Universal Robots PolyScope program: ad_lab_exe_4_2_64.urp

Program ad_lab_exe_4_2_64 (createdIn=3.2.19293 lastSavedIn=3.2.19293 directory=/programs installation=default robotSerialNumber=2015351391)
Calibrated DH parameters: a=[0.000352, -0.161198, -0.373486, 0.00005, 0.000049, 0]; d=[0.089268, 352.477598, -320.08558, -32.281492, 0.094939, 0.082518]; alpha=[1.570728, 0.001116, -0.003686, 1.571189, -1.570572, 0]; deltaTheta=[-0.000012, 1.181849, -1.491165, 0.309495, -0.000007, 0.000025]
Robot Program (runOnlyOnce=false motionType=MoveJ speed=1.047198 acceleration=1.396263 recalculateMotions=false)
  Folder 文件夹
    tcp1 := p[0,0,0.2,0,0,0]
    tcp2 := p[0.2,0,0.05,0,d2r(90),0]
    Script: set_tcp(tcp1)
    MoveL speed 250 mm/s, acceleration 1200 mm/s^2 (recalculateMotions=false) feature=Base
      Waypoint waypoint1: TCP in base x=137.871 y=664.13 z=276.516 mm, rx=-1.3493 ry=2.4374 rz=0.4077 rad; joints [96.893, -88.292, -94.384, -84.585, 94.191, -232.18] deg; flange x=46.759 y=487.114 z=417.839 mm, rx=1.522 ry=-2.6851 rz=-0.1148 rad
      Waypoint place_pos: TCP in base x=-60.021 y=25.367 z=248.738 mm, rx=0.8568 ry=-1.3626 rz=0.7366 rad; joints [108.205, -40.851, -138.273, -87.315, 93.558, -220.796] deg; flange x=46.759 y=195.075 z=296.65 mm, rx=1.522 ry=-2.6851 rz=-0.1148 rad
    Script: set_tcp(tcp2)
    offset_s1 := p[-0.075,0.075,0,0,0,0]
    offset_s2 := p[0.075,0.075,0,0,0,0]
    offset_s3 := p[-0.075,-0.075,0,0,0,0]
    offset_s4 := p[0.075,-0.075,0,0,0,0]
    screw_1 := pose_trans(place_pos,offset_s1)
    screw_2 := pose_trans(place_pos,offset_s2)
    screw_3 := pose_trans(place_pos,offset_s3)
    screw_4 := pose_trans(place_pos,offset_s4)
    MoveL speed 250 mm/s, acceleration 1200 mm/s^2 (recalculateMotions=false) feature=Base
      Waypoint relative_point1 (Relative): relativeFromPosition TCP in base x=-60.015 y=25.36 z=248.749 mm, rx=0.8567 ry=-1.3627 rz=0.7367 rad; joints [108.205, -40.851, -138.273, -87.315, 93.558, -220.796] deg; TCP in base x=-60.028 y=25.358 z=299.998 mm, rx=0.8566 ry=-1.3626 rz=0.7368 rad; joints [108.212, -41.576, -130.624, -94.244, 93.55, -220.768] deg; flange x=46.747 y=195.081 z=347.899 mm, rx=1.5221 ry=-2.6851 rz=-0.1147 rad
    MoveL speed 250 mm/s, acceleration 1200 mm/s^2 (recalculateMotions=false) feature=Base
      Waypoint 路点 (Variable): variable=screw_1
      MoveL speed 250 mm/s, acceleration 1200 mm/s^2 (recalculateMotions=false) feature=Base
        Waypoint place_pos: TCP in base x=-60.021 y=25.367 z=248.738 mm, rx=0.8568 ry=-1.3626 rz=0.7366 rad; joints [108.205, -40.851, -138.273, -87.315, 93.558, -220.796] deg; flange x=46.759 y=195.075 z=296.65 mm, rx=1.522 ry=-2.6851 rz=-0.1148 rad
      Waypoint 路点 (Variable): variable=screw_2
      MoveL speed 250 mm/s, acceleration 1200 mm/s^2 (recalculateMotions=false) feature=Base
        Waypoint place_pos: TCP in base x=-60.021 y=25.367 z=248.738 mm, rx=0.8568 ry=-1.3626 rz=0.7366 rad; joints [108.205, -40.851, -138.273, -87.315, 93.558, -220.796] deg; flange x=46.759 y=195.075 z=296.65 mm, rx=1.522 ry=-2.6851 rz=-0.1148 rad
      Waypoint 路点 (Variable): variable=screw_3
      MoveL speed 250 mm/s, acceleration 1200 mm/s^2 (recalculateMotions=false) feature=Base
        Waypoint place_pos: TCP in base x=-60.021 y=25.367 z=248.738 mm, rx=0.8568 ry=-1.3626 rz=0.7366 rad; joints [108.205, -40.851, -138.273, -87.315, 93.558, -220.796] deg; flange x=46.759 y=195.075 z=296.65 mm, rx=1.522 ry=-2.6851 rz=-0.1148 rad
      Waypoint 路点 (Variable): variable=screw_4
